Fanuc KAREL source: MP0112.KL

-- PROVISIONAL review KL for V1013-1; original PC SHA256 d18b42bc196bc649f03863d450e07d1a8abb0399cde4ad43e9e7ae9ea12872c2
-- Incomplete behavior may be omitted. Consult companion uncertainty JSON. Do not deploy.
PROGRAM MP0112
%NOLOCKGROUP
-- UNRESOLVED_LOCAL_POOL 8 cells at code offset 63; source declarations unknown
-- DIRECT_LOCAL_WORD_ACCESS alone does not prove INTEGER, REAL, or BOOLEAN
BEGIN
  -- UNRESOLVED_PC offsets 0-1; opcodes 7B
  -- UNRESOLVED_PC offsets 6-18; opcodes 2D,9D,52,7F
  -- UNRESOLVED_PC offsets 23-28; opcodes 7F,7B
  -- UNRESOLVED_PC offsets 33-49; opcodes 2D,2E,69,7F
  -- UNRESOLVED_PC offsets 54-68; opcodes 7F,2B,2C,7B
  -- UNRESOLVED_PC offsets 73-84; opcodes 2E,23
  -- UNRESOLVED_PC offsets 89-100; opcodes 2E,23
  -- UNRESOLVED_PC offsets 105-116; opcodes 2E,23
  -- UNRESOLVED_PC offsets 121-132; opcodes 2E,23
  -- UNRESOLVED_PC offsets 137-148; opcodes 2E,23
  -- UNRESOLVED_PC offsets 153-164; opcodes 2E,23
  -- UNRESOLVED_PC offsets 169-192; opcodes 22,32,34,21,6C,23
  -- UNRESOLVED_PC offsets 197-201; opcodes 7F
  -- UNRESOLVED_PC offsets 206-222; opcodes 27,27,2E,27,2E,AA
  -- UNRESOLVED_PC offsets 227-231; opcodes 7F
END MP0112
